{attribute 'qualified_only'}
{attribute 'strict'}
TYPE E_PalletDispenser :
(
	enum_member := 0
);
END_TYPE

(* stored: Version 1.1.0.1, ProductVersion 3.1.4024.12
   DUT E_PalletDispenser: Id {61626145-9403-4804-9500-d41cf6d53a02} *)
